(* IEC 61131-3 sources: Word/plc-course/04-ladder-logic/labs/starter, 4 files *)

(* ---- 04-1-start-stop-station.st ---- *)
(* Lab 04-1: Start/stop from two stations (local and remote).
   Module 04 (Ladder logic fundamentals).
   STARTER - the declarations are done for you; write the logic where it
   says TODO, then run:
     python3 tools/plctest.py 04-ladder-logic/labs/starter/04-1-start-stop-station.st
   Training exercise only: emergency stops are hard-wired or use
   safety-rated devices (Module 20). *)

PROGRAM TwoStationStart
  VAR (* I/O - addresses follow the OpenPLC convention *)
    LocalStartPB    AT %IX0.0 : BOOL;  (* Start at the local station beside the pump, NO: TRUE while pressed *)
    LocalStopPB_NC  AT %IX0.1 : BOOL;  (* Stop at the local station, NC: TRUE while NOT pressed *)
    RemoteStartPB   AT %IX0.2 : BOOL;  (* Start on the control-room panel, NO: TRUE while pressed *)
    RemoteStopPB_NC AT %IX0.3 : BOOL;  (* Stop on the control-room panel, NC: TRUE while NOT pressed *)
    Motor           AT %QX0.0 : BOOL;  (* Pump motor contactor coil *)
    RunLamp         AT %QX0.1 : BOOL;  (* "Running" lamp *)
    StoppedLamp     AT %QX0.2 : BOOL;  (* "Stopped" lamp *)
  END_VAR

  (* TODO: replace these placeholder lines with your logic.
     Sketch the ladder rung first: which contacts go in parallel, which in
     series, and which contact symbol does an NC stop button need?
     (MATIEC needs at least one statement in a program body.) *)
  Motor := FALSE;
  RunLamp := FALSE;
  StoppedLamp := FALSE;
END_PROGRAM

CONFIGURATION Config0
  RESOURCE Res0 ON PLC
    TASK MainTask(INTERVAL := T#10ms, PRIORITY := 0);
    PROGRAM Inst0 WITH MainTask : TwoStationStart;
  END_RESOURCE
END_CONFIGURATION

(* ---- 04-2-forward-reverse.st ---- *)
(* Lab 04-2: Forward/reverse motor with interlocks and travel limits.
   Module 04 (Ladder logic fundamentals).
   STARTER - the declarations are done for you; write the logic where it
   says TODO, then run:
     python3 tools/plctest.py 04-ladder-logic/labs/starter/04-2-forward-reverse.st
   A real reversing starter also has electrical and mechanical interlocks
   between its contactors. Training exercise only. *)

PROGRAM ForwardReverse
  VAR (* I/O - addresses follow the OpenPLC convention *)
    FwdPB         AT %IX0.0 : BOOL;  (* Forward push-button, NO: TRUE while pressed *)
    RevPB         AT %IX0.1 : BOOL;  (* Reverse push-button, NO: TRUE while pressed *)
    StopPB_NC     AT %IX0.2 : BOOL;  (* Stop push-button, NC: TRUE while NOT pressed *)
    FwdLimitOK_NC AT %IX0.3 : BOOL;  (* Forward end-of-travel limit switch, NC: TRUE while NOT at the limit *)
    RevLimitOK_NC AT %IX0.4 : BOOL;  (* Reverse end-of-travel limit switch, NC: TRUE while NOT at the limit *)
    OverloadOK_NC AT %IX0.5 : BOOL;  (* Overload relay auxiliary contact, NC: TRUE while healthy *)
    FwdK          AT %QX0.0 : BOOL;  (* Forward contactor coil *)
    RevK          AT %QX0.1 : BOOL;  (* Reverse contactor coil *)
  END_VAR

  (* TODO: replace these placeholder lines with your logic.
     Start from two seal-in rungs, one per direction. Then ask, for every
     contact: does it belong in the start branch or in series with the whole
     rung? Which limit switch belongs to which direction?
     (MATIEC needs at least one statement in a program body.) *)
  FwdK := FALSE;
  RevK := FALSE;
END_PROGRAM

CONFIGURATION Config0
  RESOURCE Res0 ON PLC
    TASK MainTask(INTERVAL := T#10ms, PRIORITY := 0);
    PROGRAM Inst0 WITH MainTask : ForwardReverse;
  END_RESOURCE
END_CONFIGURATION

(* ---- 04-3-jog-run.st ---- *)
(* Lab 04-3: Jog/run selector.
   Module 04 (Ladder logic fundamentals).
   STARTER - the declarations are done for you; write the logic where it
   says TODO, then run:
     python3 tools/plctest.py 04-ladder-logic/labs/starter/04-3-jog-run.st
   Training exercise only: jogging on a real machine is a safety function
   with its own rules and hardware (Modules 19 and 20). *)

PROGRAM JogRun
  VAR (* I/O - addresses follow the OpenPLC convention *)
    StartPB       AT %IX0.0 : BOOL;  (* Start push-button, NO: TRUE while pressed *)
    StopPB_NC     AT %IX0.1 : BOOL;  (* Stop push-button, NC: TRUE while NOT pressed *)
    JogPB         AT %IX0.2 : BOOL;  (* Jog push-button, NO: TRUE while pressed *)
    RunSel        AT %IX0.3 : BOOL;  (* JOG/RUN selector: TRUE = RUN, FALSE = JOG *)
    OverloadOK_NC AT %IX0.4 : BOOL;  (* Overload relay auxiliary contact, NC: TRUE while healthy *)
    Motor         AT %QX0.0 : BOOL;  (* Conveyor motor contactor coil *)
    RunLamp       AT %QX0.1 : BOOL;  (* "Running" lamp: continuous run only, not jogging *)
  END_VAR
  VAR (* internal - add any internal bits you need here *)
    Spare : BOOL;
  END_VAR

  (* TODO: replace these placeholder lines with your logic.
     Question to answer first: which bit is allowed to seal in, and is it
     the Motor output?
     (MATIEC needs at least one statement in a program body.) *)
  Motor := FALSE;
  RunLamp := FALSE;
  Spare := FALSE;
END_PROGRAM

CONFIGURATION Config0
  RESOURCE Res0 ON PLC
    TASK MainTask(INTERVAL := T#10ms, PRIORITY := 0);
    PROGRAM Inst0 WITH MainTask : JogRun;
  END_RESOURCE
END_CONFIGURATION

(* ---- 04-4-tank-fill.st ---- *)
(* Lab 04-4: Tank fill valve with set/reset (latch/unlatch).
   Module 04 (Ladder logic fundamentals).
   STARTER - the declarations are done for you; write the logic where it
   says TODO, then run:
     python3 tools/plctest.py 04-ladder-logic/labs/starter/04-4-tank-fill.st
   Training exercise only: overfill protection that matters for safety or
   the environment is a separate, independent function (Module 20). *)

PROGRAM TankFill
  VAR (* I/O - addresses follow the OpenPLC convention *)
    AutoSel        AT %IX0.0 : BOOL;  (* OFF/AUTO selector: TRUE = AUTO *)
    LevelAboveLow  AT %IX0.1 : BOOL;  (* LSL-101 low level switch: TRUE while the level is ABOVE it (switch covered) *)
    HighLevelOK_NC AT %IX0.2 : BOOL;  (* LSH-102 high level switch, NC: TRUE while the level is BELOW it; FALSE at high level or broken wire *)
    ResetPB        AT %IX0.3 : BOOL;  (* Fault reset push-button, NO: TRUE while pressed *)
    FillValve      AT %QX0.0 : BOOL;  (* XV-100 inlet valve solenoid: TRUE = open (spring return, fail closed) *)
    SensorFault    AT %QX0.1 : BOOL;  (* Amber lamp: level switches disagree (latched) *)
  END_VAR
  VAR (* internal - add what you need, for example an SR or RS instance *)
    Spare : BOOL;
  END_VAR

  (* TODO: replace these placeholder lines with your logic.
     Use a SET rung and a RESET rung for the valve (in ST: an IF that only
     writes TRUE and an IF that only writes FALSE). Which one must come last?
     (MATIEC needs at least one statement in a program body.) *)
  FillValve := FALSE;
  SensorFault := FALSE;
  Spare := FALSE;
END_PROGRAM

CONFIGURATION Config0
  RESOURCE Res0 ON PLC
    TASK MainTask(INTERVAL := T#10ms, PRIORITY := 0);
    PROGRAM Inst0 WITH MainTask : TankFill;
  END_RESOURCE
END_CONFIGURATION
